ABB RAPID module: module_WIZARD.modx

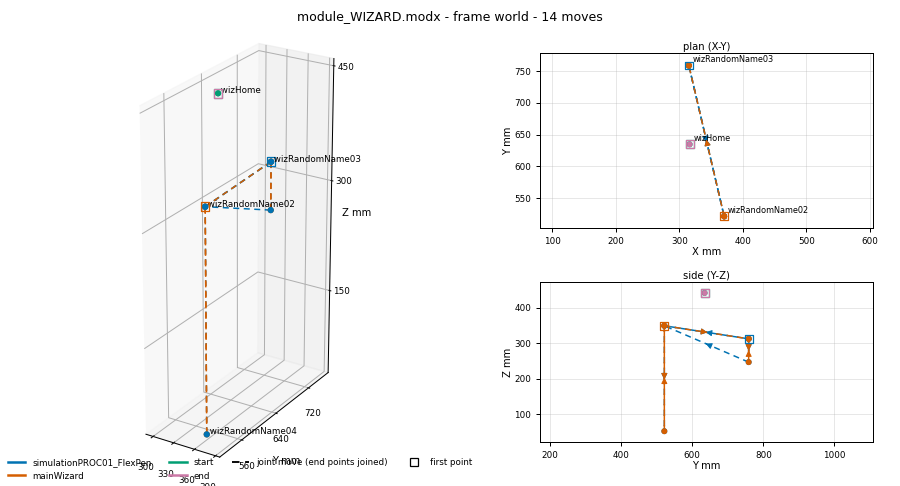
[picture p0: tool path of module_WIZARD.modx in frame world, 14 of 14 moves have a stored position in this frame; points joined in program order, loops and branches not executed]
MODULE module_WIZARD
!
!       ---------------------------------
!                   GoHolo
!       ---------------------------------
!
!       Copyright (C)   2021 Jakob Hörbst
!       author:         Jakob Hörbst
!       email:          jakob@hoerbst.net
!       year:           2021
!

PERS robtarget wizHome:=[[316.17333984375, 634.73046875, 440.990356445313], [0.0026820998173207, 0.00783746875822544, 0.999948501586914, 0.00585808232426643], [0, 0, 0, 0], [9000000000, 9000000000, 9000000000, 9000000000, 9000000000, 9000000000]];
PERS robtarget wizRandomName02:=[[370.495269775391, 521.374877929688, 348.593353271484], [0.00379902473650873, 0.701789557933807, 0.712373673915863, -0.000882733904290944], [0, -1, 1, 0], [9000000000, 9000000000, 9000000000, 9000000000, 9000000000, 9000000000]];
PERS robtarget wizRandomName04:=[[370.480529785156, 521.381530761719, 51.8949508666992], [0.00380251440219581, 0.708827674388885, 0.705370903015137, -0.000862757791765034], [0, -1, 1, 0], [9000000000, 9000000000, 9000000000, 9000000000, 9000000000, 9000000000]];
PERS robtarget wizRandomName03:=[[314.93212890625, 758.710083007813, 311.827056884766], [0.00269204052165151, 0.00783240702003241, 0.999948382377625, 0.00589012308046222], [0, -1, 0, 0], [9000000000, 9000000000, 9000000000, 9000000000, 9000000000, 9000000000]];
PERS robtarget wizRandomName01:=[[314.909301757813, 758.708068847656, 246.256469726563], [0.00268639274872839, 0.00781508535146713, 0.999948561191559, 0.00588054535910487], [0, -1, 0, 0], [9000000000, 9000000000, 9000000000, 9000000000, 9000000000, 9000000000]];
PERS robtarget wizRandomName11:=[[370.495269775391, 521.374877929688, 348.593353271484], [0.00379902473650873, 0.701789557933807, 0.712373673915863, -0.000882733904290944], [0, -1, 1, 0], [9000000000, 9000000000, 9000000000, 9000000000, 9000000000, 9000000000]];
PERS robtarget wizRandomName13:=[[370.480529785156, 521.381530761719, 51.8949508666992], [0.00380251440219581, 0.708827674388885, 0.705370903015137, -0.000862757791765034], [0, -1, 1, 0], [9000000000, 9000000000, 9000000000, 9000000000, 9000000000, 9000000000]];
PERS robtarget wizRandomName14:=[[314.93212890625, 758.710083007813, 311.827056884766], [0.00269204052165151, 0.00783240702003241, 0.999948382377625, 0.00589012308046222], [0, -1, 0, 0], [9000000000, 9000000000, 9000000000, 9000000000, 9000000000, 9000000000]];
PERS robtarget wizRandomName12:=[[314.909301757813, 758.708068847656, 246.256469726563], [0.00268639274872839, 0.00781508535146713, 0.999948561191559, 0.00588054535910487], [0, -1, 0, 0], [9000000000, 9000000000, 9000000000, 9000000000, 9000000000, 9000000000]];
PROC simulationPROC01_FlexPendant()
    start;
    MoveJ wizRandomName03, v100, fine, tool0;
    MoveJ wizRandomName02, v100, fine, tool0;
    MoveJ wizRandomName03, v100, fine, tool0;
    MoveJ wizRandomName01, v100, fine, tool0;
    MoveJ wizRandomName02, v100, fine, tool0;
    MoveJ wizRandomName04, v100, fine, tool0;
    end;
ENDPROC
PROC mainWizard()
start;
MoveJ wizRandomName11, v100, fine, tool0;
MoveJ wizRandomName13, v100, fine, tool0;
MoveJ wizRandomName11, v100, fine, tool0;
MoveJ wizRandomName14, v100, fine, tool0;
MoveJ wizRandomName12, v100, fine, tool0;
MoveJ wizRandomName14, v100, fine, tool0;
end;
ENDPROC
PROC simulationPROC02_HoloLens2()
ENDPROC
PROC start()
    MoveJ wizHome, v200, fine, tool0;
ENDPROC
PROC end()
    MoveJ wizHome, v200, fine, tool0;
ENDPROC
ENDMODULE
